ABB RobotStudio station: TEST1.rsstn

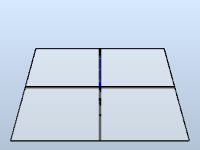
Station TEST1 (saved by RobotStudio 6.8.8148.134)
Controller IRB_120_3kg_0.58m
  mechanical unit ROB_1: ?, 6 joints, base frame (0, 0, 0) mm
Layout (positions relative to the parent item):
